// TIA Portal V17 export
// export: Created 2024-08-29T18:23:50.5133359Z, ExportSetting WithDefaults, DisplayName Totally Integrated Automation Portal, DisplayVersion V17 Update 7, DisplayName TIA Portal Openness, DisplayVersion V17 Update 7, DisplayName TIA Portal Version Control Interface, DisplayVersion V17, DisplayName SINAMICS Startdrive Advanced, DisplayVersion V17 SP2, DisplayName SINAMICS Startdrive G110M, G120, G120C, G120D, G120P, G115D, DisplayVersion V17 SP2, DisplayName SINAMICS Startdrive G130, G150, S120, S150, SINAMICS MV, S210, DisplayVersion V17 SP2, DisplayName STEP 7 Professional, DisplayVersion V17 Update 7, DisplayName STEP 7 Safety, DisplayVersion V17 Update 6, DisplayName WinCC Advanced / Unified PC, DisplayVersion V17 Update 7
VAR_GLOBAL   // PLC tag table "DCmotorControlMemory"
   motorBackwardMotion AT %M1551.2 : Bool;
   motorForwardMotion AT %M1550.7 : Bool;
   motorOpposite AT %M1551.4 : Bool;
   motorMovementActive AT %M1550.6 : Bool;
   hmiTestLeftMotorAlignment AT %M1551.6 : Bool;
   hmiTestRightTrackAlignment AT %M1551.7 : Bool;
   motorDirection AT %M1550.4 : Bool;
   highPulseDone AT %M1550.5 : Bool;
   reset AT %M1552.0 : Bool;
   direction1Pulse AT %MW1500 : Int;
   ctuReset1 AT %M1550.3 : Bool;
   motorPulseWidthSelector AT %M1551.5 : Bool;
   motorPulseWIidth AT %MD1534 : DInt;
   motorCycleTime AT %MD1530 : DInt;
   motorPulseQuantity AT %MW1502 : Int;
   activateMotorOperation AT %M1550.0 : Bool;
   hmiMoveMotorForward AT %M1552.1 : Bool;
   hmiMoveMotorBackward AT %M1552.2 : Bool;
   moveMotorForward AT %M1550.1 : Bool;
   moveMotorBackward AT %M1550.2 : Bool;
   leftTrackAlignmentComplete AT %M1551.1 : Bool;
   rightTrackAlignmentComplete AT %M1551.0 : Bool;
END_VAR
